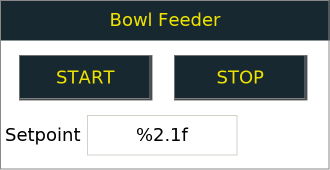
VISUALIZATION AOIBowlFeederFrame  // 330x170
    Rectangle (0,0 330x40), "Bowl Feeder"
    Button (19,55 133x45), "START"
        tap PRG_MachineControl.fbMachineControler.btnStartBowl
    Textfield (87,115 150x40), "%2.1f", text variable: PRG_MachineControl.fbMachineControler.rBowlFeederSetpoint
        OnMouseClick: write the text variable via VisuDialogs.Numpad
    Label (2,120 98x30), "Setpoint"
    Button (174,55 133x45), "STOP"
        tap PRG_MachineControl.fbMachineControler.btnStopBowl
END_VISUALIZATION

(* stored: Version 1.1.0.1, ProductVersion 3.1.4024.9
   Visu AOIBowlFeederFrame: Id {583ee471-59dd-4d00-a947-cd79525c7b53} *)
